# EPICS alarm handler configuration: mps_database/bare/alarms/areas/mpln_l0b_mp02.alhConfig
GROUP NULL MPLN:L0B:MP02:1
$ALIAS MPS Link Node 52
$GUIDANCE
LTUH MPS
   Group Name: MPLN:L0B:MP02:1
   Summary PV:  MPLN:L0B:MP02:1:STATSUMY
$END
CHANNEL  MPLN:L0B:MP02:1    MPLN:L0B:MP02:1:MPS_EN_RBV		-----
CHANNEL  MPLN:L0B:MP02:1    MPLN:L0B:MP02:1:LC1_MODE_RBV		-----
